Fanuc KAREL source: GET_FILE_POS.kl

PROGRAM T
%NOLOCKGROUP
VAR
 v0 : FILE
 res : INTEGER
BEGIN
 res = GET_FILE_POS(v0)
END T
